PROGRAM MAIN
VAR
	//cmt 1
	bTest_1 : BOOL;
END_VAR

// --- Version 1 --- 
// Program 1
// -----------------

END_PROGRAM

(* stored: Version 1.1.0.1, ProductVersion 3.1.4024.10
   POU MAIN: Id {51aa1b40-096d-43e9-9fc4-b34a7ff3d064}, SpecialFunc None *)
